(* IEC 61131-3 sources: Industry-PLC-LLM/data/PLCBEAD_repo/PLCBEAD_PLCEmbed-main/PLC-BEAD/Source/GEB/MIN3, 1 file *)

(* ---- MIN3.ST ---- *)
FUNCTION MIN3:REAL

	VAR_INPUT
		IN1 :	REAL;
		IN2 :	REAL;
		IN3 :	REAL;
	END_VAR

	MIN3 := MIN(MIN(IN1,IN2),IN3);

END_FUNCTION

PROGRAM program0

	VAR
		IN1 :	REAL;
		IN2 :	REAL;
		IN3 :	REAL;
		CEIL5_OUT : REAL;
	END_VAR

	CEIL5_OUT := MIN3(IN1, IN2, IN3);

END_PROGRAM
